PROGRAM Main
VAR

	Hour_Meter : Hour_Meter_FB;


	TempVar : BOOL := TRUE;
	
	poop: STRING;
	connected : Bool;
END_VAR

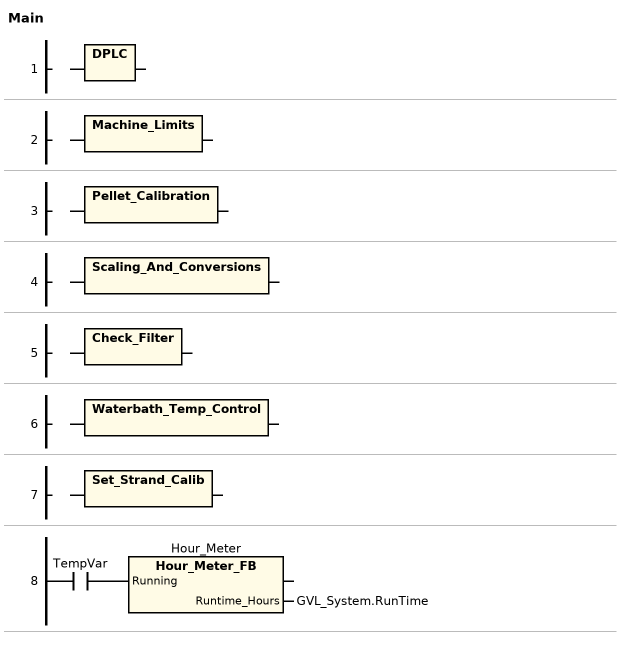
// NETWORK 1
DPLC();

// NETWORK 2
Machine_Limits();

// NETWORK 3
Pellet_Calibration();

// NETWORK 4
Scaling_And_Conversions();

// NETWORK 5
Check_Filter();

// NETWORK 6
Waterbath_Temp_Control();

// NETWORK 7
Set_Strand_Calib();

// NETWORK 8
Hour_Meter(Running := TempVar, Runtime_Hours => GVL_System.RunTime); // Hour_Meter_FB

END_PROGRAM

(* stored: Version 1.1.0.1, ProductVersion 3.1.4024.12
   POU Main: Id {2ad019de-d0a4-4668-a92c-2ee0c996bdad}, SpecialFunc None *)
